# EPICS substitutions: ioc/bsdaq.substitutions
file bsdaq.template {
	pattern{P} {BSREAD}
}
